(* CoDeSys 2.3.9.50 project: 4C.pr6 *)
(* Libraries: STANDARD.LB6 5.6.98 12:03:02 *)

(* POU MAIN, LD *)
PROGRAM MAIN
VAR
	A AT %IX0.0: BOOL;
	B AT %IX0.1: BOOL;
	C AT %IX0.2: BOOL;
	D AT %IX0.3: BOOL;
	CA: CTU;
	CB: CTD;
	CC: CTU;
	CD: CTD;
	L AT %QX0.0: BOOL;
	M AT %QX0.1: BOOL;
	N AT %QX0.2: BOOL;
	MasterON AT %IX0.7: BOOL;
	reset AT %IX0.6: BOOL;
	MasterReset AT %QX0.4: BOOL;
END_VAR
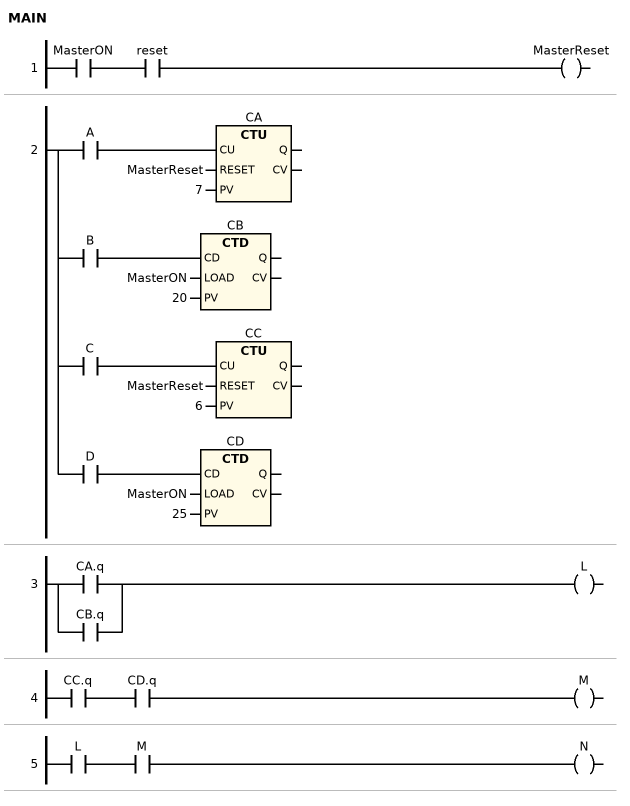
_LD_ (* Ladder Diagram *)
NETWORK 1
	[MasterON] - [reset] --- (MasterReset)
NETWORK 2
	{ [A] - CA:CTU(CU: *, RESET: MasterReset, PV: 7) | [B] - CB:CTD(CD: *, LOAD: MasterON, PV: 20) | [C] - CC:CTU(CU: *, RESET: MasterReset, PV: 6) | [D] - CD:CTD(CD: *, LOAD: MasterON, PV: 25) }
NETWORK 3
	{ [CA.q] | [CB.q] } --- (L)
NETWORK 4
	[CC.q] - [CD.q] --- (M)
NETWORK 5
	[L] - [M] --- (N)
_END_LD_
(* the same logic as Structured Text *)
(* Network 1 *)
MasterReset := MasterON AND reset;
(* Network 2 *)
CA(CU := A, RESET := MasterReset, PV := 7);
CB(CD := B, LOAD := MasterON, PV := 20);
CC(CU := C, RESET := MasterReset, PV := 6);
CD(CD := D, LOAD := MasterON, PV := 25);
(* Network 3 *)
L := CA.q OR CB.q;
(* Network 4 *)
M := CC.q AND CD.q;
(* Network 5 *)
N := L AND M;
END_PROGRAM
